SUBAPPLICATION Uebung_160b (* Motor Links/Rechtslauf Automatisierung via IE *)
  (* Standard: 61499-2; Description: Copyright (c) 2023 Meisterschulen am Ostbahnhof This program and the accompanying materials are made available under the terms of the Eclipse Public License 2.0 which is available at https://www.eclipse.org/legal/epl-2.0/ SPDX-License-Identifier: EPL-2.0 *)
  (* Version 1.1, 2026-04-19, Franz Höpfinger, Meisterschulen am Ostbahnhof, Cleaned imports and improved FB naming *)
  PACKAGE Uebungen;
  IMPORT logiBUS::io::DI::logiBUS_DI::Input_I1;
  IMPORT logiBUS::io::DI::logiBUS_DI::Input_I2;
  IMPORT logiBUS::io::DI::logiBUS_DI::Input_I3;
  IMPORT logiBUS::io::DI::logiBUS_DI_Events::BUTTON_PRESS_DOWN;
  IMPORT logiBUS::io::DI::logiBUS_DI_Events::BUTTON_SINGLE_CLICK;
  IMPORT logiBUS::io::DQ::logiBUS_DO::Output_Q5;
  IMPORT logiBUS::io::DQ::logiBUS_DO::Output_Q6;
  IMPORT logiBUS::io::DQ::logiBUS_DO::Output_Q56;
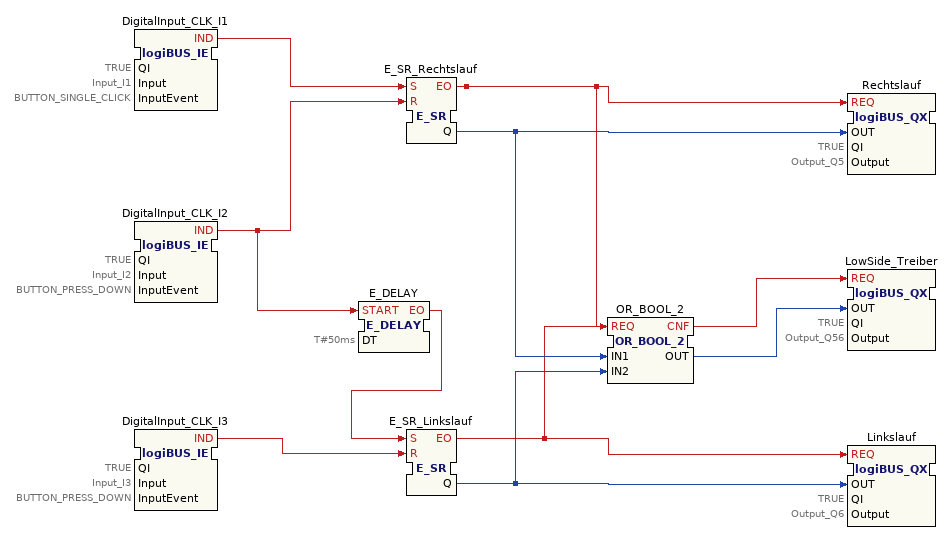
  FBS
    Linkslauf : logiBUS::io::DQ::logiBUS_QX(QI := TRUE, Output := Output_Q6);
    E_SR_Linkslauf : iec61499::events::E_SR;
    OR_BOOL_2 : iec61131::booleanOperators::OR_BOOL_2;
    E_SR_Rechtslauf : iec61499::events::E_SR;
    Rechtslauf : logiBUS::io::DQ::logiBUS_QX(QI := TRUE, Output := Output_Q5);
    LowSide_Treiber : logiBUS::io::DQ::logiBUS_QX(QI := TRUE, Output := Output_Q56);
    DigitalInput_CLK_I2 : logiBUS::io::DI::logiBUS_IE(QI := TRUE, Input := Input_I2, InputEvent := BUTTON_PRESS_DOWN);
    DigitalInput_CLK_I3 : logiBUS::io::DI::logiBUS_IE(QI := TRUE, Input := Input_I3, InputEvent := BUTTON_PRESS_DOWN);
    DigitalInput_CLK_I1 : logiBUS::io::DI::logiBUS_IE(QI := TRUE, Input := Input_I1, InputEvent := BUTTON_SINGLE_CLICK);
    E_DELAY : iec61499::events::E_DELAY(DT := T#50ms);
  END_FBS
  EVENT_CONNECTIONS
    E_SR_Linkslauf.EO TO Linkslauf.REQ;
    E_SR_Rechtslauf.EO TO Rechtslauf.REQ;
    OR_BOOL_2.CNF TO LowSide_Treiber.REQ;
    E_SR_Linkslauf.EO TO OR_BOOL_2.REQ;
    E_SR_Rechtslauf.EO TO OR_BOOL_2.REQ;
    DigitalInput_CLK_I1.IND TO E_SR_Rechtslauf.S;
    DigitalInput_CLK_I2.IND TO E_SR_Rechtslauf.R;
    DigitalInput_CLK_I2.IND TO E_DELAY.START;
    E_DELAY.EO TO E_SR_Linkslauf.S;
    DigitalInput_CLK_I3.IND TO E_SR_Linkslauf.R;
  END_CONNECTIONS
  DATA_CONNECTIONS
    E_SR_Linkslauf.Q TO Linkslauf.OUT;
    E_SR_Rechtslauf.Q TO Rechtslauf.OUT;
    OR_BOOL_2.OUT TO LowSide_Treiber.OUT;
    E_SR_Rechtslauf.Q TO OR_BOOL_2.IN1;
    E_SR_Linkslauf.Q TO OR_BOOL_2.IN2;
  END_CONNECTIONS
END_SUBAPPLICATION
